{region '#Template'}
	{attribute 'Version' := '6.1.0.0'}
	{attribute 'Tags' := '"LCID": "1031", "Text": "AC, Setpoint, Temperatur, Cascade control"'}
	{attribute 'Tags' := '"LCID": "1033", "Text": "AC, Setpoint, Temperatur, Cascade control"'}
	{attribute 'Using' := '"Type": "Template", "URI": "Priority"'}		 
	{attribute 'Using' := '"Type": "Template", "URI": "BA2_Param"'}
	{attribute 'Description' := '"LCID": "1031", "Text": "Temperatur Kaskadenregelung"'}
	{attribute 'Description' := '"LCID": "1033", "Text": "Temperature Cascade control"'}
{endregion}
FUNCTION_BLOCK FB_BA_AC_TCasCtrl_01 EXTENDS FB_BA_View
VAR_INPUT
	fSpTRm					: REAL;
	fTRm					: REAL;
END_VAR                                                         	
VAR_OUTPUT                                                      	
	fSpHtg					: REAL;
	fSpCol					: REAL;
	fSpErc					: REAL;
	fMax					: REAL;
	fMin					: REAL;
	bOn						: BOOL;	
END_VAR
VAR_IN_OUT
	stAggregate				: ST_BA_Aggregate;	
END_VAR
VAR_INPUT CONSTANT
	Sp						: FB_BA_AV_Op;									
	Ctrl					: FB_BA_Loop;	
	Aggregate				: FB_BA_Aggregate;																											 								
END_VAR
VAR
	PrioSwiVal				: FB_BA_PrioSwi_UDI04;	
	MuxCmd					: FB_BA_MMUX_B04;	
	MuxSp					: FB_BA_MMUX_R04;
END_VAR

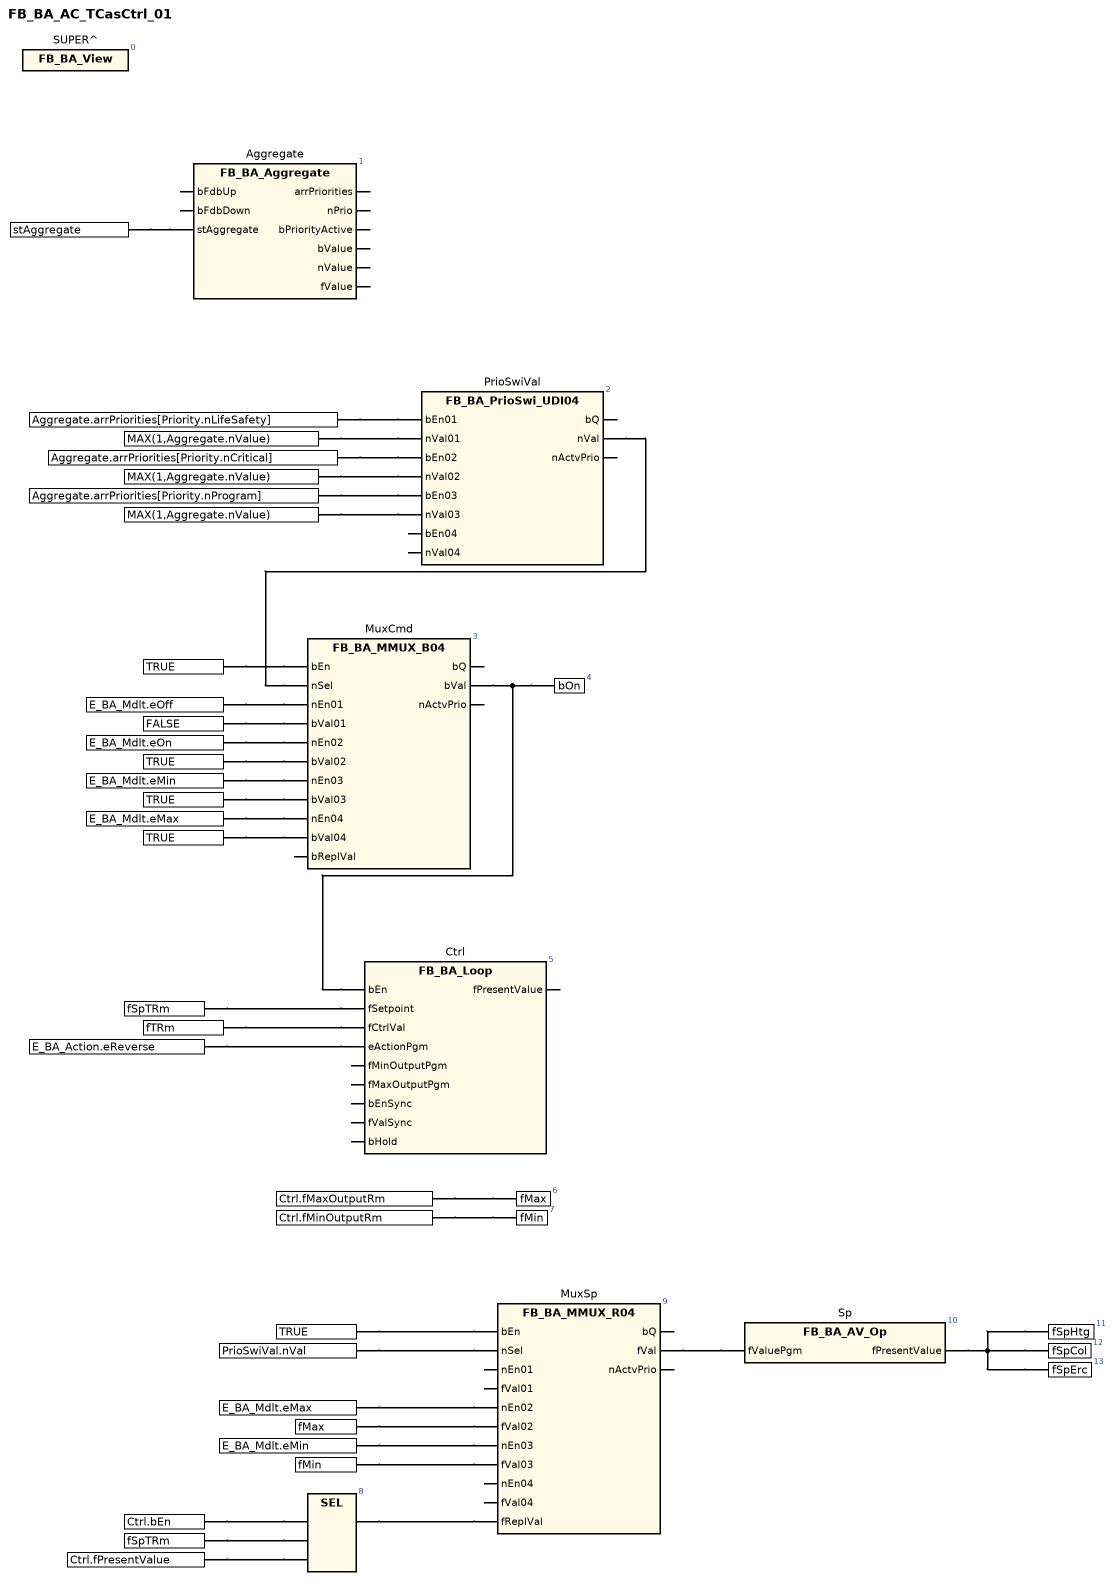
SUPER^(); // FB_BA_View
Aggregate(stAggregate := stAggregate); // FB_BA_Aggregate
PrioSwiVal(
    bEn01 := Aggregate.arrPriorities[Priority.nLifeSafety],
    nVal01 := MAX(1,Aggregate.nValue),
    bEn02 := Aggregate.arrPriorities[Priority.nCritical],
    nVal02 := MAX(1,Aggregate.nValue),
    bEn03 := Aggregate.arrPriorities[Priority.nProgram],
    nVal03 := MAX(1,Aggregate.nValue)); // FB_BA_PrioSwi_UDI04
MuxCmd(
    bEn := TRUE,
    nSel := PrioSwiVal.nVal,
    nEn01 := E_BA_Mdlt.eOff,
    bVal01 := FALSE,
    nEn02 := E_BA_Mdlt.eOn,
    bVal02 := TRUE,
    nEn03 := E_BA_Mdlt.eMin,
    bVal03 := TRUE,
    nEn04 := E_BA_Mdlt.eMax,
    bVal04 := TRUE); // FB_BA_MMUX_B04
bOn := MuxCmd.bVal;
Ctrl(bEn := MuxCmd.bVal, fSetpoint := fSpTRm, fCtrlVal := fTRm, eActionPgm := E_BA_Action.eReverse); // FB_BA_Loop
fMax := Ctrl.fMaxOutputRm;
fMin := Ctrl.fMinOutputRm;
MuxSp(
    bEn := TRUE,
    nSel := PrioSwiVal.nVal,
    nEn02 := E_BA_Mdlt.eMax,
    fVal02 := fMax,
    nEn03 := E_BA_Mdlt.eMin,
    fVal03 := fMin,
    fReplVal := SEL(Ctrl.bEn, fSpTRm, Ctrl.fPresentValue)); // FB_BA_MMUX_R04
Sp(fValuePgm := MuxSp.fVal); // FB_BA_AV_Op
fSpHtg := Sp.fPresentValue;
fSpCol := Sp.fPresentValue;
fSpErc := Sp.fPresentValue;

METHOD FB_init : BOOL
VAR_INPUT
	bInitRetains : BOOL; // if TRUE, the retain variables are initialized (warm start / cold start)
	bInCopyCode : BOOL;  // if TRUE, the instance afterwards gets moved into the copy code (online change)
END_VAR
Sp.iParent						:= THIS^;
Sp.iLabel						:= LblCtl_SuppyAirTempSetpointCalc; 				 	 
Sp.eUnit							:= E_BA_Unit.eTemperature_DegreesCelsius;  
Sp.fCOVIncrement					:= BA2_Param.fDefCOVIncrement;							

Ctrl.iParent						:= THIS^;
Ctrl.iLabel							:= LblFun_LoopObjectCascadeSupplyAirTemperature; 	
Ctrl.eOpMode						:= E_BA_PIDMode.ePID;							 	 										 
Ctrl.eOutputUnit					:= E_BA_Unit.eTemperature_DegreesCelsius;
Ctrl.fProportionalConstant			:= 3;
Ctrl.fIntegralConstant				:= 180;
Ctrl.fDerivativeConstant			:= 0;
Ctrl.fMaxOutputRm 					:= 32;
Ctrl.fMinOutputRm					:= 16;
Ctrl.fCOVIncrement					:= 0;
Ctrl.nDampConstant					:= 0;
Ctrl.fNeutralZone					:= 0;
END_METHOD

END_FUNCTION_BLOCK

(* stored: Version 1.1.0.1, ProductVersion 3.1.4024.15
   POU FB_BA_AC_TCasCtrl_01: Id {bc1a9304-2d21-4853-bfb6-7def207edbc7}, SpecialFunc None
   Method FB_init: Id {384a0b3e-897d-4d36-96e9-6ad8e9b68cda} *)
